SUBAPPLICATION InputOutputTesterBt_OPC_UA (* Tester *)
  (* Standard: 61499-2; Description: Copyright (c) 2023 Meisterschulen am Ostbahnhof This program and the accompanying materials are made available under the terms of the Eclipse Public License 2.0 which is available at https://www.eclipse.org/legal/epl-2.0/ SPDX-License-Identifier: EPL-2.0 *)
  (* Version 1.0, 2023-10-23, Franz Höpfinger, Meisterschulen am Ostbahnhof, initial API and implementation and/or initial documentation *)
  PACKAGE Meins;
  IMPORT Uebungen::const::UT::Tester::DefaultPool_Tester::Button_I01;
  IMPORT Uebungen::const::UT::Tester::DefaultPool_Tester::Button_I02;
  IMPORT Uebungen::const::UT::Tester::DefaultPool_Tester::Button_I03;
  IMPORT Uebungen::const::UT::Tester::DefaultPool_Tester::Button_I04;
  IMPORT Uebungen::const::UT::Tester::DefaultPool_Tester::Button_I05;
  IMPORT Uebungen::const::UT::Tester::DefaultPool_Tester::Button_I06;
  IMPORT Uebungen::const::UT::Tester::DefaultPool_Tester::Button_I07;
  IMPORT Uebungen::const::UT::Tester::DefaultPool_Tester::Button_I08;
  IMPORT Uebungen::const::UT::Tester::DefaultPool_Tester::Button_Q01;
  IMPORT Uebungen::const::UT::Tester::DefaultPool_Tester::Button_Q02;
  IMPORT Uebungen::const::UT::Tester::DefaultPool_Tester::Button_Q03;
  IMPORT Uebungen::const::UT::Tester::DefaultPool_Tester::Button_Q04;
  IMPORT Uebungen::const::UT::Tester::DefaultPool_Tester::Button_Q05;
  IMPORT Uebungen::const::UT::Tester::DefaultPool_Tester::Button_Q06;
  IMPORT Uebungen::const::UT::Tester::DefaultPool_Tester::Button_Q07;
  IMPORT Uebungen::const::UT::Tester::DefaultPool_Tester::Button_Q08;
  IMPORT Uebungen::const::UT::Tester::DefaultPool_Tester::Button_Q09;
  IMPORT Uebungen::const::UT::Tester::DefaultPool_Tester::Button_Q10;
  IMPORT Uebungen::const::UT::Tester::DefaultPool_Tester::Button_Q11;
  IMPORT Uebungen::const::UT::Tester::DefaultPool_Tester::Button_Q12;
  IMPORT logiBUS::io::DQ::logiBUS_DO;
  IMPORT logiBUS::io::DI::logiBUS_DI;
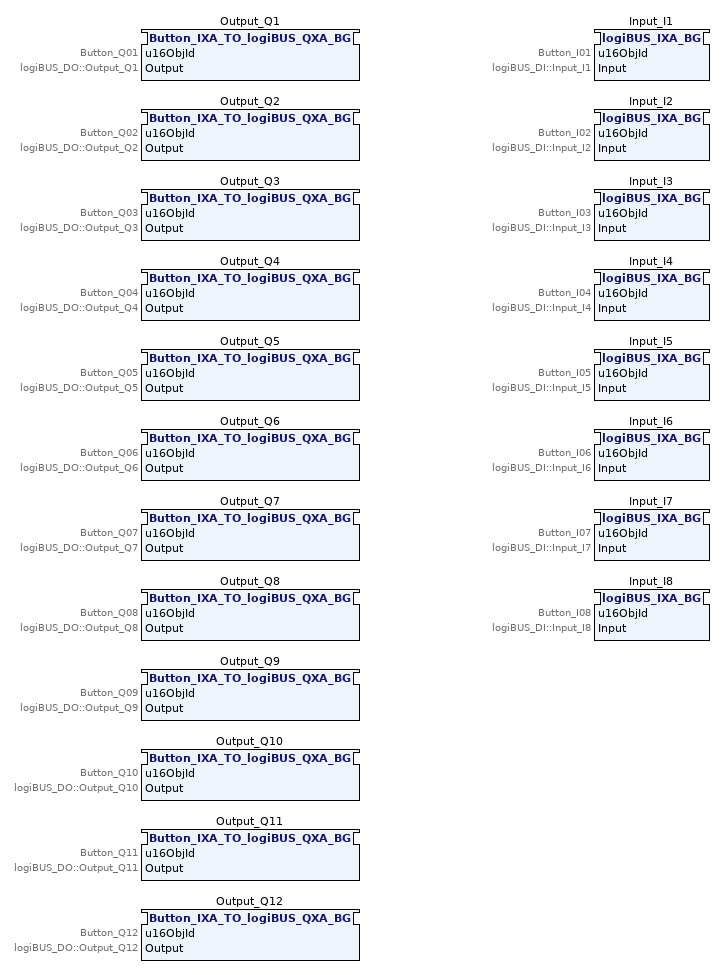
  SUBAPPS
    Input_I1 : MyLib::sys::logiBUS_IXA_BG(u16ObjId := Button_I01, Input := logiBUS_DI::Input_I1);
    Input_I2 : MyLib::sys::logiBUS_IXA_BG(u16ObjId := Button_I02, Input := logiBUS_DI::Input_I2);
    Input_I3 : MyLib::sys::logiBUS_IXA_BG(u16ObjId := Button_I03, Input := logiBUS_DI::Input_I3);
    Input_I4 : MyLib::sys::logiBUS_IXA_BG(u16ObjId := Button_I04, Input := logiBUS_DI::Input_I4);
    Input_I5 : MyLib::sys::logiBUS_IXA_BG(u16ObjId := Button_I05, Input := logiBUS_DI::Input_I5);
    Input_I6 : MyLib::sys::logiBUS_IXA_BG(u16ObjId := Button_I06, Input := logiBUS_DI::Input_I6);
    Input_I7 : MyLib::sys::logiBUS_IXA_BG(u16ObjId := Button_I07, Input := logiBUS_DI::Input_I7);
    Input_I8 : MyLib::sys::logiBUS_IXA_BG(u16ObjId := Button_I08, Input := logiBUS_DI::Input_I8);
    Output_Q1 : MyLib::sys::Button_IXA_TO_logiBUS_QXA_BG(u16ObjId := Button_Q01, Output := logiBUS_DO::Output_Q1);
    Output_Q2 : MyLib::sys::Button_IXA_TO_logiBUS_QXA_BG(u16ObjId := Button_Q02, Output := logiBUS_DO::Output_Q2);
    Output_Q3 : MyLib::sys::Button_IXA_TO_logiBUS_QXA_BG(u16ObjId := Button_Q03, Output := logiBUS_DO::Output_Q3);
    Output_Q4 : MyLib::sys::Button_IXA_TO_logiBUS_QXA_BG(u16ObjId := Button_Q04, Output := logiBUS_DO::Output_Q4);
    Output_Q5 : MyLib::sys::Button_IXA_TO_logiBUS_QXA_BG(u16ObjId := Button_Q05, Output := logiBUS_DO::Output_Q5);
    Output_Q6 : MyLib::sys::Button_IXA_TO_logiBUS_QXA_BG(u16ObjId := Button_Q06, Output := logiBUS_DO::Output_Q6);
    Output_Q7 : MyLib::sys::Button_IXA_TO_logiBUS_QXA_BG(u16ObjId := Button_Q07, Output := logiBUS_DO::Output_Q7);
    Output_Q8 : MyLib::sys::Button_IXA_TO_logiBUS_QXA_BG(u16ObjId := Button_Q08, Output := logiBUS_DO::Output_Q8);
    Output_Q9 : MyLib::sys::Button_IXA_TO_logiBUS_QXA_BG(u16ObjId := Button_Q09, Output := logiBUS_DO::Output_Q9);
    Output_Q10 : MyLib::sys::Button_IXA_TO_logiBUS_QXA_BG(u16ObjId := Button_Q10, Output := logiBUS_DO::Output_Q10);
    Output_Q11 : MyLib::sys::Button_IXA_TO_logiBUS_QXA_BG(u16ObjId := Button_Q11, Output := logiBUS_DO::Output_Q11);
    Output_Q12 : MyLib::sys::Button_IXA_TO_logiBUS_QXA_BG(u16ObjId := Button_Q12, Output := logiBUS_DO::Output_Q12);
  END_SUBAPPS
END_SUBAPPLICATION
